(* IEC 61131-3 sources: SPSZL-PLC-DenOD/SinKarusel/KaruselPas1, 1 file *)

(* ---- prgMain.ST ---- *)
PROGRAM prgMain
  VAR
  END_VAR

  pojezd := NOT(vyrobekPodChnap);

END_PROGRAM
